{attribute addProperty BoxType "KL1032"}
{attribute addProperty Id "Channel_1Channel_70B606D100Channel_2Channel_70B606D100"}
{attribute addProperty CRC "3525945802"}
{attribute addProperty SizeInBites "0"}
{attribute addProperty SizeInBytes "0"}
TYPE KL1032_D229A9CA :
STRUCT
	{attribute addProperty Name "Channel_1"}
	Channel_1 : Channel_70B606D1;
	{attribute addProperty Name "Channel_2"}
	Channel_2 : Channel_70B606D1;
END_STRUCT
END_TYPE

(* stored: Version 1.2.0.0, ProductVersion 3.1.4024.9
   DUT KL1032_D229A9CA: Id {54c58e2d-4bf8-4290-a433-2b2133cda2b5} *)
